PROGRAM MAIN
VAR
	
	fbZAFan			 : FB_ZA_Fan;
END_VAR


fbZAFan();

END_PROGRAM

(* stored: Version 1.1.0.1, ProductVersion 3.1.4024.12
   POU MAIN: Id {ffecc0be-3ece-405c-bd0b-1ec36ceb0d51}, SpecialFunc None *)
